Fanuc KAREL source: kb00166.KL

-- PROVISIONAL review KL for V1013-1; original PC SHA256 9367cb6aa2c51fc90bc2eed90c1d381a1638f493c01ace267fafde964364ec02
-- Incomplete behavior may be omitted. Consult companion uncertainty JSON. Do not deploy.
PROGRAM KB00166
%NOLOCKGROUP
BEGIN
  -- UNRESOLVED_PC offsets 5-12; opcodes 9D,23
  -- UNRESOLVED_PC offsets 17-24; opcodes 9D,23
  -- UNRESOLVED_PC offsets 29-59; opcodes 27,22,22,1C,22,27,9D,31
  -- UNRESOLVED_PC offsets 64-68; opcodes 7F
END KB00166
